% RSLogix 500 project 2_PUMP_SYS_BAK008.RSS, saved by version 8.30.00.16 %
PROJECT "UNTITLED"    % processor: Bul.1763 MicroLogix 1100 Series B %

PROGRAM FILES
  LAD 2   7 rungs
  LAD 3 "PUMP 1"  5 rungs
  LAD 4 "PUMP 2"  5 rungs
  LAD 5 "IN VLV 1"  2 rungs
  LAD 6 "IN VLV 2"  2 rungs
  LAD 7 "RECIRC VLV"  2 rungs
  LAD 8 "SCHEDULING"  8 rungs
  LAD 9 "ALMS"  1 rungs

DATA FILES
  O0 OUTPUT  4 elements
  I1 INPUT  6 elements
  S2 STATUS  66 elements
  B3 BINARY  12 elements
  T4 TIMER  20 elements
  C5 COUNTER  1 elements
  R6 CONTROL  1 elements
  N7 INTEGER  1 elements
  F8 FLOAT  1 elements

LADDER 2
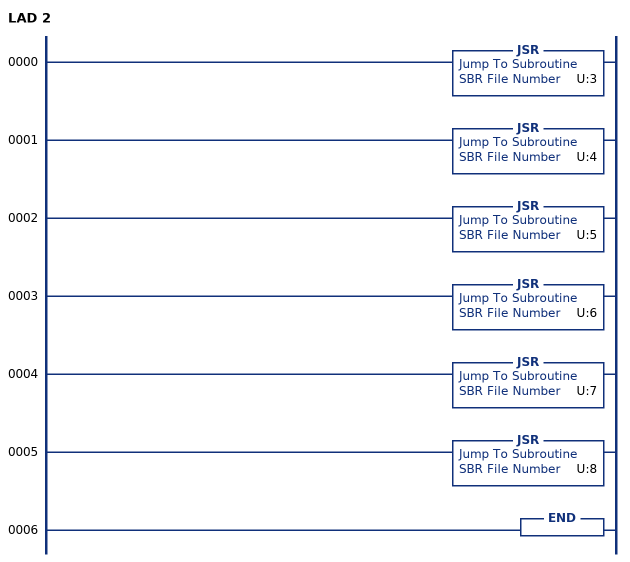
% Rung: 0 %
SOR JSR U:3 EOR
% Rung: 1 %
SOR JSR U:4 EOR
% Rung: 2 %
SOR JSR U:5 EOR
% Rung: 3 %
SOR JSR U:6 EOR
% Rung: 4 %
SOR JSR U:7 EOR
% Rung: 5 %
SOR JSR U:8 EOR
% Rung: 6 %
SOR END EOR

LADDER 3 "PUMP 1"
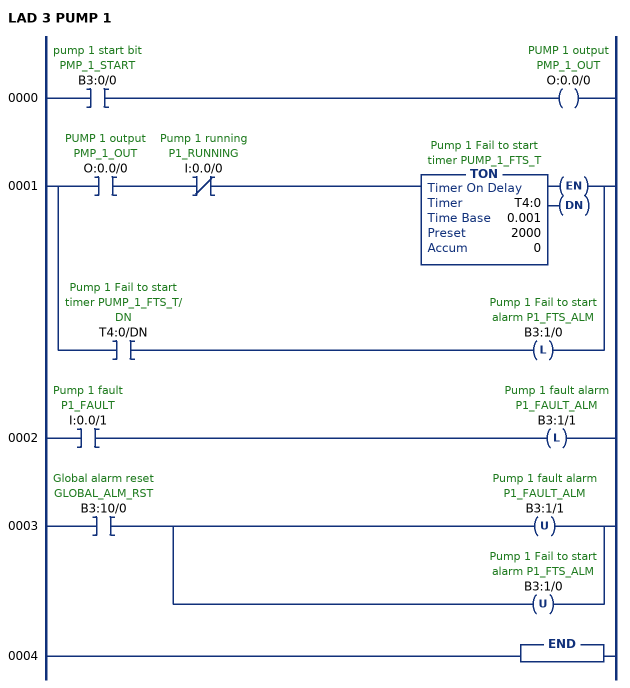
% Rung: 0 %
SOR XIC B3:0/0 OTE O:0.0/0 EOR
%   B3:0/0  PMP_1_START  "pump 1 start bit" %
%   O:0.0/0  PMP_1_OUT  "PUMP 1 output" %
% Rung: 1 %
SOR BST XIC O:0.0/0 XIO I:0.0/0 TON T4:0 0.001 2000 0 NXB XIC T4:0/DN OTL B3:1/0 BND EOR
%   O:0.0/0  PMP_1_OUT  "PUMP 1 output" %
%   I:0.0/0  P1_RUNNING  "Pump 1 running" %
%   T4:0  PUMP_1_FTS_T  "Pump 1 Fail to start timer" %
%   B3:1/0  P1_FTS_ALM  "Pump 1 Fail to start alarm" %
% Rung: 2 %
SOR XIC I:0.0/1 OTL B3:1/1 EOR
%   I:0.0/1  P1_FAULT  "Pump 1 fault" %
%   B3:1/1  P1_FAULT_ALM  "Pump 1 fault alarm" %
% Rung: 3 %
SOR XIC B3:10/0 BST OTU B3:1/1 NXB OTU B3:1/0 BND EOR
%   B3:10/0  GLOBAL_ALM_RST  "Global alarm reset" %
%   B3:1/1  P1_FAULT_ALM  "Pump 1 fault alarm" %
%   B3:1/0  P1_FTS_ALM  "Pump 1 Fail to start alarm" %
% Rung: 4 %
SOR END EOR

LADDER 4 "PUMP 2"
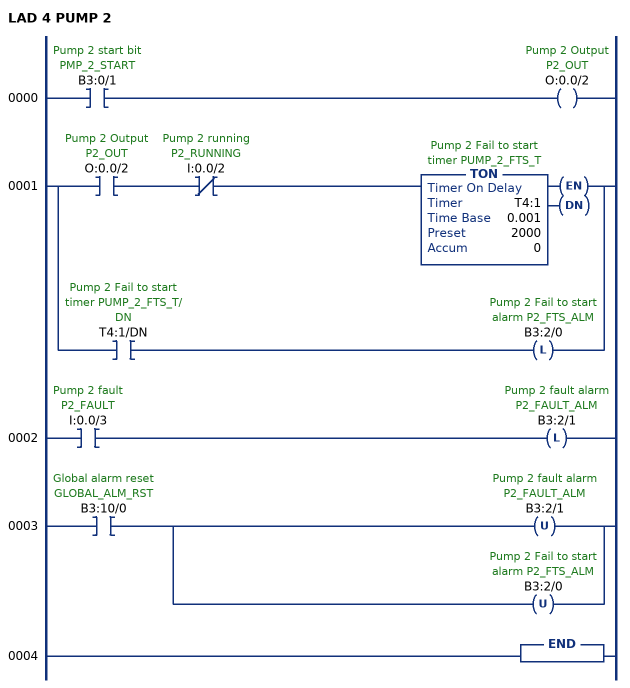
% Rung: 0 %
SOR XIC B3:0/1 OTE O:0.0/2 EOR
%   B3:0/1  PMP_2_START  "Pump 2 start bit" %
%   O:0.0/2  P2_OUT  "Pump 2 Output" %
% Rung: 1 %
SOR BST XIC O:0.0/2 XIO I:0.0/2 TON T4:1 0.001 2000 0 NXB XIC T4:1/DN OTL B3:2/0 BND EOR
%   O:0.0/2  P2_OUT  "Pump 2 Output" %
%   I:0.0/2  P2_RUNNING  "Pump 2 running" %
%   T4:1  PUMP_2_FTS_T  "Pump 2 Fail to start timer" %
%   B3:2/0  P2_FTS_ALM  "Pump 2 Fail to start alarm" %
% Rung: 2 %
SOR XIC I:0.0/3 OTL B3:2/1 EOR
%   I:0.0/3  P2_FAULT  "Pump 2 fault" %
%   B3:2/1  P2_FAULT_ALM  "Pump 2 fault alarm" %
% Rung: 3 %
SOR XIC B3:10/0 BST OTU B3:2/1 NXB OTU B3:2/0 BND EOR
%   B3:10/0  GLOBAL_ALM_RST  "Global alarm reset" %
%   B3:2/1  P2_FAULT_ALM  "Pump 2 fault alarm" %
%   B3:2/0  P2_FTS_ALM  "Pump 2 Fail to start alarm" %
% Rung: 4 %
SOR END EOR

LADDER 5 "IN VLV 1"
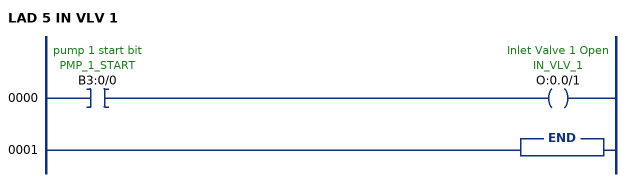
% Rung: 0 %
SOR XIC B3:0/0 OTE O:0.0/1 EOR
%   B3:0/0  PMP_1_START  "pump 1 start bit" %
%   O:0.0/1  IN_VLV_1  "Inlet Valve 1 Open" %
% Rung: 1 %
SOR END EOR

LADDER 6 "IN VLV 2"
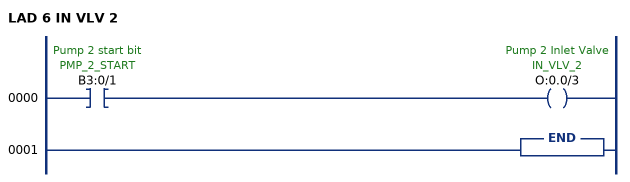
% Rung: 0 %
SOR XIC B3:0/1 OTE O:0.0/3 EOR
%   B3:0/1  PMP_2_START  "Pump 2 start bit" %
%   O:0.0/3  IN_VLV_2  "Pump 2 Inlet Valve" %
% Rung: 1 %
SOR END EOR

LADDER 7 "RECIRC VLV"
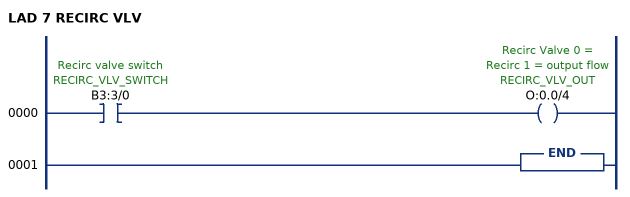
% Rung: 0 %
SOR XIC B3:3/0 OTE O:0.0/4 EOR
%   B3:3/0  RECIRC_VLV_SWITCH  "Recirc valve switch" %
%   O:0.0/4  RECIRC_VLV_OUT  "Recirc Valve 0 = Recirc 1 = output flow" %
% Rung: 1 %
SOR END EOR

LADDER 8 "SCHEDULING"
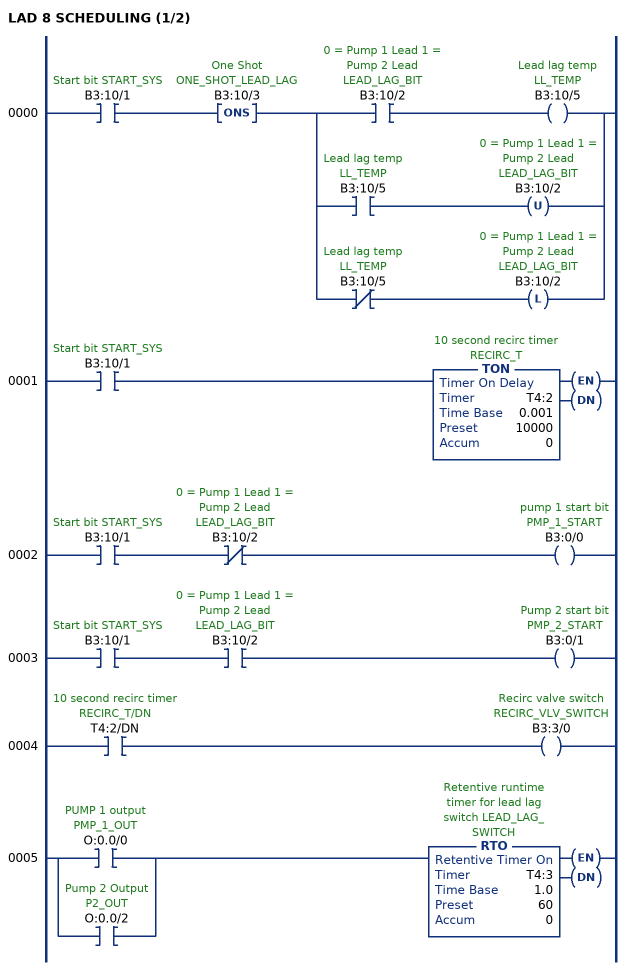
% Rung: 0 %
SOR XIC B3:10/1 ONS B3:10/3 BST BST XIC B3:10/2 OTE B3:10/5 NXB XIC B3:10/5 OTU B3:10/2 BND NXB XIO B3:10/5 OTL B3:10/2 BND EOR
%   B3:10/1  START_SYS  "Start bit" %
%   B3:10/3  ONE_SHOT_LEAD_LAG  "One Shot" %
%   B3:10/2  LEAD_LAG_BIT  "0 = Pump 1 Lead 1 = Pump 2 Lead" %
%   B3:10/5  LL_TEMP  "Lead lag temp" %
% Rung: 1 %
SOR XIC B3:10/1 TON T4:2 0.001 10000 0 EOR
%   B3:10/1  START_SYS  "Start bit" %
%   T4:2  RECIRC_T  "10 second recirc timer" %
% Rung: 2 %
SOR XIC B3:10/1 XIO B3:10/2 OTE B3:0/0 EOR
%   B3:10/1  START_SYS  "Start bit" %
%   B3:10/2  LEAD_LAG_BIT  "0 = Pump 1 Lead 1 = Pump 2 Lead" %
%   B3:0/0  PMP_1_START  "pump 1 start bit" %
% Rung: 3 %
SOR XIC B3:10/1 XIC B3:10/2 OTE B3:0/1 EOR
%   B3:10/1  START_SYS  "Start bit" %
%   B3:10/2  LEAD_LAG_BIT  "0 = Pump 1 Lead 1 = Pump 2 Lead" %
%   B3:0/1  PMP_2_START  "Pump 2 start bit" %
% Rung: 4 %
SOR XIC T4:2/DN OTE B3:3/0 EOR
%   T4:2  RECIRC_T  "10 second recirc timer" %
%   B3:3/0  RECIRC_VLV_SWITCH  "Recirc valve switch" %
% Rung: 5 %
SOR BST XIC O:0.0/0 NXB XIC O:0.0/2 BND RTO T4:3 1.0 60 0 EOR
%   O:0.0/0  PMP_1_OUT  "PUMP 1 output" %
%   O:0.0/2  P2_OUT  "Pump 2 Output" %
%   T4:3  LEAD_LAG_SWITCH  "Retentive runtime timer for lead lag switch" %

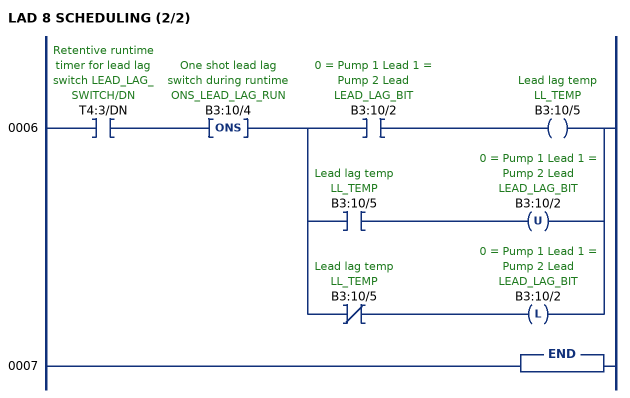
% Rung: 6 %
SOR XIC T4:3/DN ONS B3:10/4 BST BST XIC B3:10/2 OTE B3:10/5 NXB XIC B3:10/5 OTU B3:10/2 BND NXB XIO B3:10/5 OTL B3:10/2 BND EOR
%   T4:3  LEAD_LAG_SWITCH  "Retentive runtime timer for lead lag switch" %
%   B3:10/4  ONS_LEAD_LAG_RUN  "One shot lead lag switch during runtime" %
%   B3:10/2  LEAD_LAG_BIT  "0 = Pump 1 Lead 1 = Pump 2 Lead" %
%   B3:10/5  LL_TEMP  "Lead lag temp" %
% Rung: 7 %
SOR END EOR

DATA TABLE (non-zero values as saved)
DATA B3
% B3:10 % 0X0004 0X0000
DATA T4
% .PRE .ACC %
% T4:0 % 2000 0
% T4:1 % 2000 0
% T4:2 % 10000 0
% T4:3 % 60 0
